// TIA Portal V20 export
TYPE "ROUT_Destino_Desvios"
   STRUCT
      Destino : UInt;   // Destino de la Etiqueta
      Desvios : Array[0.."ROUT_Num_Max_Desvios"] of Struct   // Desvios por las Etiquetas
         SCR : UInt;   // Numero de SCR
         Bits : Byte;   // Bits a Activar
         Libre : Byte;   // Byte libre para opciones a añadir en la estructura sin que crezca
      END_STRUCT;
   END_STRUCT;
   // Desvios[0..20].Bits := B#16#01;
END_TYPE
